PROGRAM MAIN
VAR
	fbPV : FB_Hoymiles_DTU_ProS_PV_Inverter;

END_VAR

	
					
fbPV(
	bEnable:= , 
	sIPAdress:= '192.168.1.216', 
	byUnitID_Inverter:= 101, 
	DataHoymiles_DTU_Pro_Total=> , 
	arrDataHoymiles_DTU_Pro=> , 
	stDataEMPower_PV=> , 
	stDataEMCounter_PV=> , 
	diNrOfEM_OUT_PV=> );

END_PROGRAM

(* stored: Version 1.1.0.1, ProductVersion 3.1.4024.11
   POU MAIN: Id {c3d880a7-a386-488f-8782-4173f050ebd2}, SpecialFunc None *)
